// TIA Portal V16 export
// export: Created 2023-03-29T11:04:29.3880965Z, ExportSetting WithDefaults, DisplayName Totally Integrated Automation Portal, DisplayVersion V16 Update 6, DisplayName TIA Portal Version Control Interface, DisplayVersion V16 Update 2, DisplayName TIA Portal Openness, DisplayVersion V16 Update 6, DisplayName STEP 7 Professional, DisplayVersion V16 Update 6, DisplayName STEP 7 Safety, DisplayVersion V16, DisplayName WinCC Advanced, DisplayVersion V16 Update 6
FUNCTION_BLOCK "VLV02"   // FB5, LAD
TITLE = Valve driver 02
{ S7_Optimized_Access := 'FALSE' }
AUTHOR : RTecmer
VERSION : 0.2
// Driver for two-position drives
// Slowo STATUSU Napedu
// STAT - Prawy Byte
// WIZ  - Lewy Byte
//  
//   -STAT wektor stanu zaworu
//     -bit 0- alarm                                  (sygnal do SCADA)
//     -bit 1- zawor otwarty                    (sygnal do SCADA)
//     -bit 2-sterowanie zdal=1 loc=0 (sygnal do SCADA)
//     -bit 3- zawor zamkniety               (sygnal do SCADA)
//     -bit 4-otwieranie reczne              (sygnal z SCADA)
//     -bit 5-zamykanie reczne              (sygnal z SCADA)
//     -bit 6-alarm reset                        (sygnal z SCADA
//     -bit 8-auto= 1man=0                  (sygnal z SCADA)
//   -SUPV 
//   -CLSD zawor zamkniety                    - wejscie
//   -OPND zawor otwarty                        - wejscie
//   -REMT sterowanie zdal=1 loc=0      - wejscie
//   -OPEN otwarcie                                  - wyjscie
//   -CLSE zamkniecie                              - wyjscie
//   - TIM1 czas otwierania  
//   - TIM2 czas zamykania
// stored: AutoNumber true, IsIECCheckEnabled false, SetENOAutomatically false, UDAEnableTagReadback false
   VAR_INPUT
      SVMC : Bool;   // Automat na zamykanie
      SVMO { ExternalVisible := 'False'} : Bool;   // Automat na otwieranie
      CLSD : Bool;   // Zamknięta
      OPND : Bool;   // Otwarta
      REMT : Bool;   // Sterowanie zdalne =1, remontowe=0
      KT1 : Time;   // Czas timera
   END_VAR
   VAR_IN_OUT
      CLSE { ExternalAccessible := 'False'; ExternalVisible := 'False'; ExternalWritable := 'False'} : Bool;   // Wyjście zamykanie
      OPEN { ExternalAccessible := 'False'; ExternalVisible := 'False'; ExternalWritable := 'False'} : Bool;   // Wyjście Otwieranie
      WIZ : Byte;   // Wektor SCADA
      STAT : Byte;   // Wektor statusu napędu
      TMR1 : TON_TIME;
   END_VAR
BEGIN

REGION Network 1
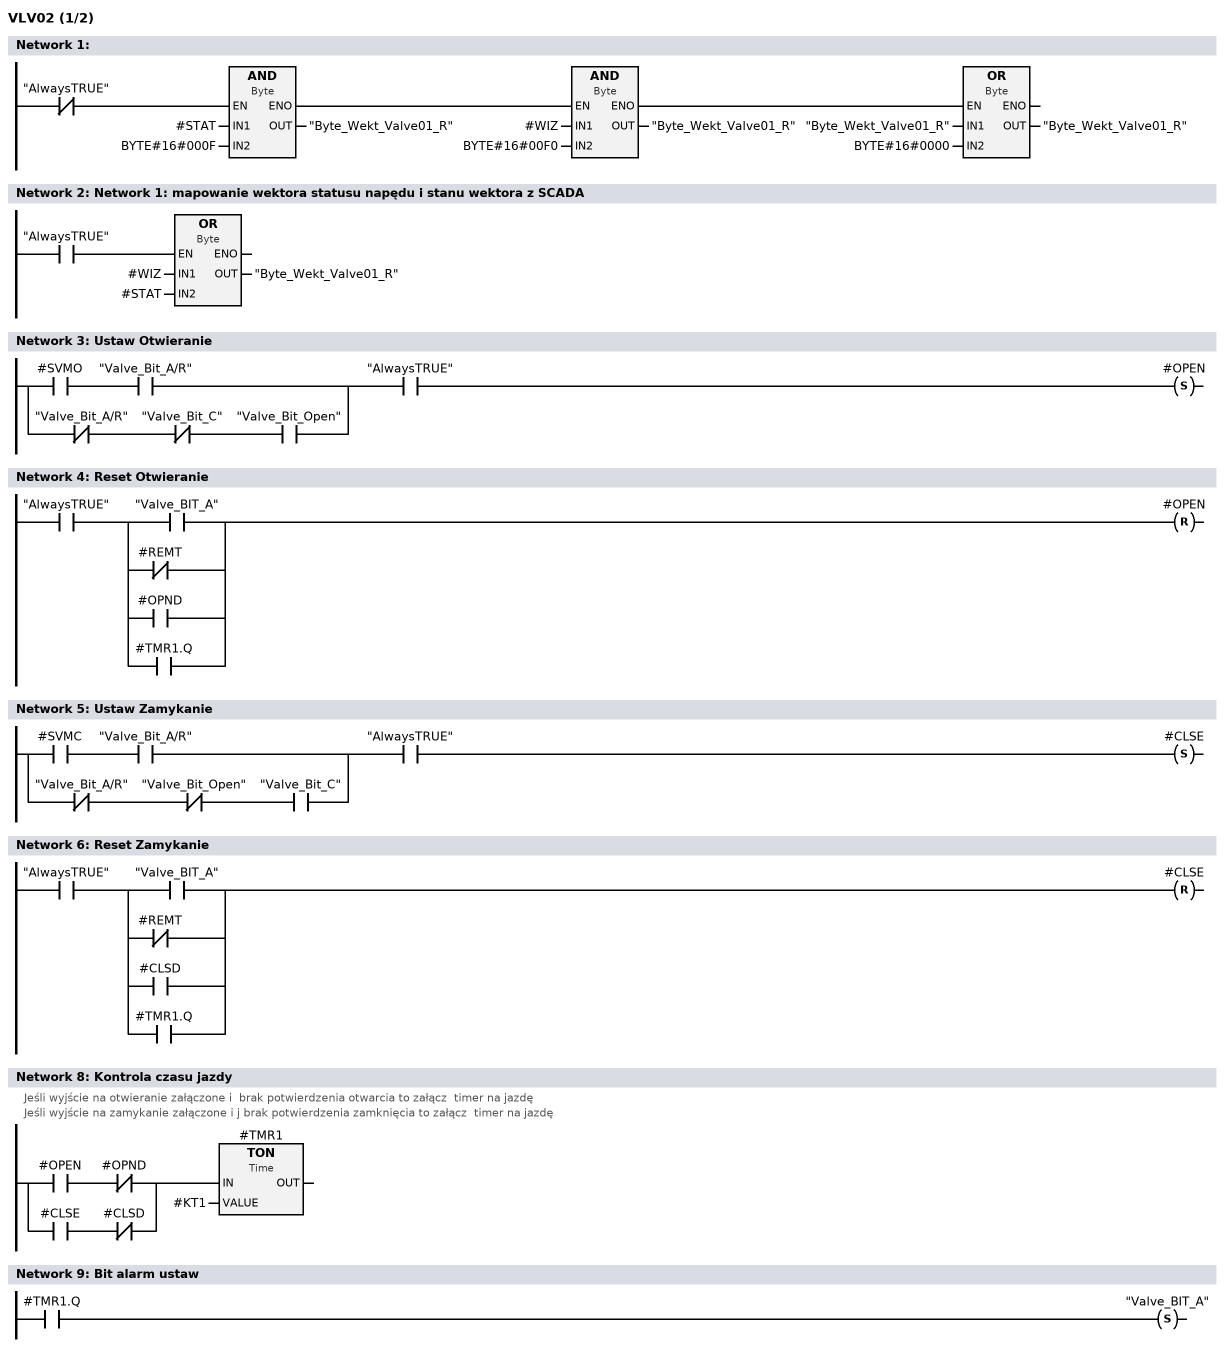
   IF NOT "AlwaysTRUE" THEN
       "Byte_Wekt_Valve01_R" := #STAT AND BYTE#16#000F;
       "Byte_Wekt_Valve01_R" := #WIZ AND BYTE#16#00F0;
       "Byte_Wekt_Valve01_R" := "Byte_Wekt_Valve01_R" OR BYTE#16#0000;
   END_IF;
END_REGION

REGION Network 2: Network 1: mapowanie wektora statusu napędu i stanu wektora z SCADA
   IF "AlwaysTRUE" THEN "Byte_Wekt_Valve01_R" := #WIZ OR #STAT; END_IF;
END_REGION

REGION Network 3: Ustaw Otwieranie
   RUNG wire#powerrail
      Contact( #SVMO )
      Contact( "Valve_Bit_A/R" )
      wire#w1
      Contact( "AlwaysTRUE" )
      S_Coil( #OPEN )
   END_RUNG
   RUNG wire#powerrail
      I_Contact( "Valve_Bit_A/R" )
      I_Contact( "Valve_Bit_C" )
      Contact( "Valve_Bit_Open" )
   END_RUNG wire#w1
   // the same network as SCL:
   IF ((#SVMO AND "Valve_Bit_A/R") OR (NOT "Valve_Bit_A/R" AND NOT "Valve_Bit_C" AND "Valve_Bit_Open")) AND "AlwaysTRUE" THEN
       #OPEN := TRUE;
   END_IF;
END_REGION

REGION Network 4: Reset Otwieranie
   RUNG wire#powerrail
      Contact( "AlwaysTRUE" )
      wire#w1
      Contact( "Valve_BIT_A" )
      wire#w2
      R_Coil( #OPEN )
   END_RUNG
   RUNG wire#w1
      I_Contact( #REMT )
   END_RUNG wire#w2
   RUNG wire#w1
      Contact( #OPND )
   END_RUNG wire#w2
   RUNG wire#w1
      Contact( #TMR1.Q )
   END_RUNG wire#w2
   // the same network as SCL:
   IF "AlwaysTRUE" AND ("Valve_BIT_A" OR NOT #REMT OR #OPND OR #TMR1.Q) THEN #OPEN := FALSE; END_IF;
END_REGION

REGION Network 5: Ustaw Zamykanie
   RUNG wire#powerrail
      Contact( #SVMC )
      Contact( "Valve_Bit_A/R" )
      wire#w1
      Contact( "AlwaysTRUE" )
      S_Coil( #CLSE )
   END_RUNG
   RUNG wire#powerrail
      I_Contact( "Valve_Bit_A/R" )
      I_Contact( "Valve_Bit_Open" )
      Contact( "Valve_Bit_C" )
   END_RUNG wire#w1
   // the same network as SCL:
   IF ((#SVMC AND "Valve_Bit_A/R") OR (NOT "Valve_Bit_A/R" AND NOT "Valve_Bit_Open" AND "Valve_Bit_C")) AND "AlwaysTRUE" THEN
       #CLSE := TRUE;
   END_IF;
END_REGION

REGION Network 6: Reset Zamykanie
   RUNG wire#powerrail
      Contact( "AlwaysTRUE" )
      wire#w1
      Contact( "Valve_BIT_A" )
      wire#w2
      R_Coil( #CLSE )
   END_RUNG
   RUNG wire#w1
      I_Contact( #REMT )
   END_RUNG wire#w2
   RUNG wire#w1
      Contact( #CLSD )
   END_RUNG wire#w2
   RUNG wire#w1
      Contact( #TMR1.Q )
   END_RUNG wire#w2
   // the same network as SCL:
   IF "AlwaysTRUE" AND ("Valve_BIT_A" OR NOT #REMT OR #CLSD OR #TMR1.Q) THEN #CLSE := FALSE; END_IF;
END_REGION

REGION Network 8: Kontrola czasu jazdy
   // Jeśli wyjście na otwieranie załączone i  brak potwierdzenia otwarcia to załącz  timer na jazdę
   // Jeśli wyjście na zamykanie załączone i j brak potwierdzenia zamknięcia to załącz  timer na jazdę
   #TMR1(IN := (#OPEN AND NOT #OPND) OR (#CLSE AND NOT #CLSD), PT := #KT1);   // TON coil
END_REGION

REGION Network 9: Bit alarm ustaw
   RUNG wire#powerrail
      Contact( #TMR1.Q )
      S_Coil( "Valve_BIT_A" )
   END_RUNG
   // the same network as SCL:
   IF #TMR1.Q THEN "Valve_BIT_A" := TRUE; END_IF;
END_REGION

REGION Network 10: Kasowanie Bitu alarmu
   // znacznik (normalnie zwarty) #TMR1.Q  - usunięty
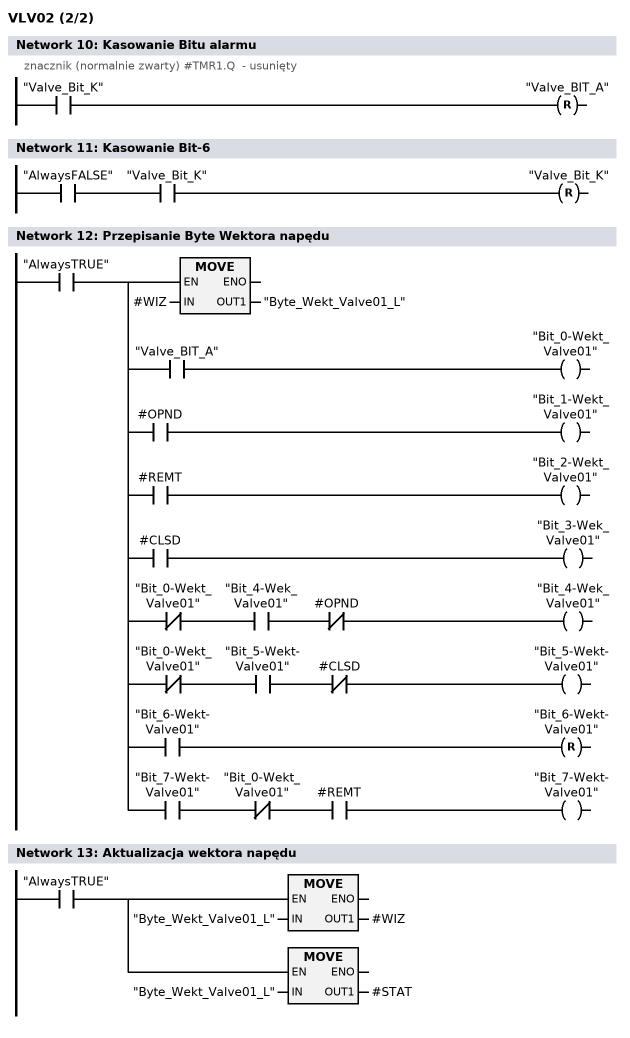
   RUNG wire#powerrail
      Contact( "Valve_Bit_K" )
      R_Coil( "Valve_BIT_A" )
   END_RUNG
   // the same network as SCL:
   IF "Valve_Bit_K" THEN "Valve_BIT_A" := FALSE; END_IF;
END_REGION

REGION Network 11: Kasowanie Bit-6
   RUNG wire#powerrail
      Contact( "AlwaysFALSE" )
      Contact( "Valve_Bit_K" )
      R_Coil( "Valve_Bit_K" )
   END_RUNG
   // the same network as SCL:
   IF "AlwaysFALSE" AND "Valve_Bit_K" THEN "Valve_Bit_K" := FALSE; END_IF;
END_REGION

REGION Network 12: Przepisanie Byte Wektora napędu
   RUNG wire#powerrail
      Contact( "AlwaysTRUE" )
      wire#w1
      { S7_GenerateENO := "TRUE" } Move(in := #WIZ, out1 => "Byte_Wekt_Valve01_L")
   END_RUNG
   RUNG wire#w1
      Contact( "Valve_BIT_A" )
      Coil( "Bit_0-Wekt_Valve01" )
   END_RUNG
   RUNG wire#w1
      Contact( #OPND )
      Coil( "Bit_1-Wekt_Valve01" )
   END_RUNG
   RUNG wire#w1
      Contact( #REMT )
      Coil( "Bit_2-Wekt_Valve01" )
   END_RUNG
   RUNG wire#w1
      Contact( #CLSD )
      Coil( "Bit_3-Wek_Valve01" )
   END_RUNG
   RUNG wire#w1
      I_Contact( "Bit_0-Wekt_Valve01" )
      Contact( "Bit_4-Wek_Valve01" )
      I_Contact( #OPND )
      Coil( "Bit_4-Wek_Valve01" )
   END_RUNG
   RUNG wire#w1
      I_Contact( "Bit_0-Wekt_Valve01" )
      Contact( "Bit_5-Wekt-Valve01" )
      I_Contact( #CLSD )
      Coil( "Bit_5-Wekt-Valve01" )
   END_RUNG
   RUNG wire#w1
      Contact( "Bit_6-Wekt-Valve01" )
      R_Coil( "Bit_6-Wekt-Valve01" )
   END_RUNG
   RUNG wire#w1
      Contact( "Bit_7-Wekt-Valve01" )
      I_Contact( "Bit_0-Wekt_Valve01" )
      Contact( #REMT )
      Coil( "Bit_7-Wekt-Valve01" )
   END_RUNG
   // the same network as SCL:
   IF "AlwaysTRUE" THEN "Byte_Wekt_Valve01_L" := #WIZ; END_IF;
   "Bit_0-Wekt_Valve01" := "AlwaysTRUE" AND "Valve_BIT_A";
   "Bit_1-Wekt_Valve01" := "AlwaysTRUE" AND #OPND;
   "Bit_2-Wekt_Valve01" := "AlwaysTRUE" AND #REMT;
   "Bit_3-Wek_Valve01" := "AlwaysTRUE" AND #CLSD;
   "Bit_4-Wek_Valve01" := "AlwaysTRUE" AND NOT "Bit_0-Wekt_Valve01" AND "Bit_4-Wek_Valve01" AND NOT #OPND;
   "Bit_5-Wekt-Valve01" := "AlwaysTRUE" AND NOT "Bit_0-Wekt_Valve01" AND "Bit_5-Wekt-Valve01" AND NOT #CLSD;
   IF "AlwaysTRUE" AND "Bit_6-Wekt-Valve01" THEN "Bit_6-Wekt-Valve01" := FALSE; END_IF;
   "Bit_7-Wekt-Valve01" := "AlwaysTRUE" AND "Bit_7-Wekt-Valve01" AND NOT "Bit_0-Wekt_Valve01" AND #REMT;
END_REGION

REGION Network 13: Aktualizacja wektora napędu
   RUNG wire#powerrail
      Contact( "AlwaysTRUE" )
      wire#w1
      { S7_GenerateENO := "TRUE" } Move(in := "Byte_Wekt_Valve01_L", out1 => #WIZ)
   END_RUNG
   RUNG wire#w1
      { S7_GenerateENO := "TRUE" } Move(in := "Byte_Wekt_Valve01_L", out1 => #STAT)
   END_RUNG
   // the same network as SCL:
   IF "AlwaysTRUE" THEN
       #WIZ := "Byte_Wekt_Valve01_L";
       #STAT := "Byte_Wekt_Valve01_L";
   END_IF;
END_REGION
END_FUNCTION_BLOCK
